FUNCTION_BLOCK RetriggerEvent (* Composite Function Block Type *)
  (* Standard: 61499-2 *)
  (* Version 0.0, 6/24/2026, Schneider Electric, template *)
  PACKAGE SE.Nereda;
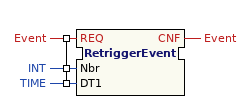
  EVENT_INPUT
    REQ WITH Nbr, DT1; (* Normal Execution Request *)
  END_EVENT
  EVENT_OUTPUT
    CNF; (* Execution Confirmation *)
  END_EVENT
  VAR_INPUT
    Nbr : INT; (* Input event qualifier *)
    DT1 : TIME; (* Delay Time *)
  END_VAR
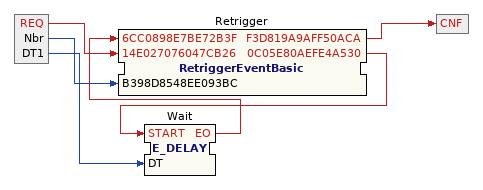
  FBS
    Wait : E_DELAY;
    Retrigger : RetriggerEventBasic;
  END_FBS
  EVENT_CONNECTIONS
    Retrigger.F3D819A9AFF50ACA TO CNF;
    Retrigger.0C05E80AEFE4A530 TO Wait.START;
    Wait.EO TO Retrigger.6CC0898E7BE72B3F;
    REQ TO Retrigger.14E027076047CB26;
  END_CONNECTIONS
  DATA_CONNECTIONS
    DT1 TO Wait.DT;
    Nbr TO Retrigger.B398D8548EE093BC;
  END_CONNECTIONS
END_FUNCTION_BLOCK
